(* CoDeSys 2.3 export: NEWARRAY.EXP *)

(* POU NewArray, ST *)
FUNCTION NewArray : POINTER TO BYTE
VAR_INPUT
	ArrayLength : Length;		(*Количество элементов в массиве*)
	ElementSize : Size;		(*Размер элемента массива в байтах*)
END_VAR
VAR
	p: POINTER TO ArrayOfByte;
END_VAR
p:= SysMemAlloc(ArrayLength*ElementSize);
p^.length := ArrayLength;
NewArray := p;
END_FUNCTION
